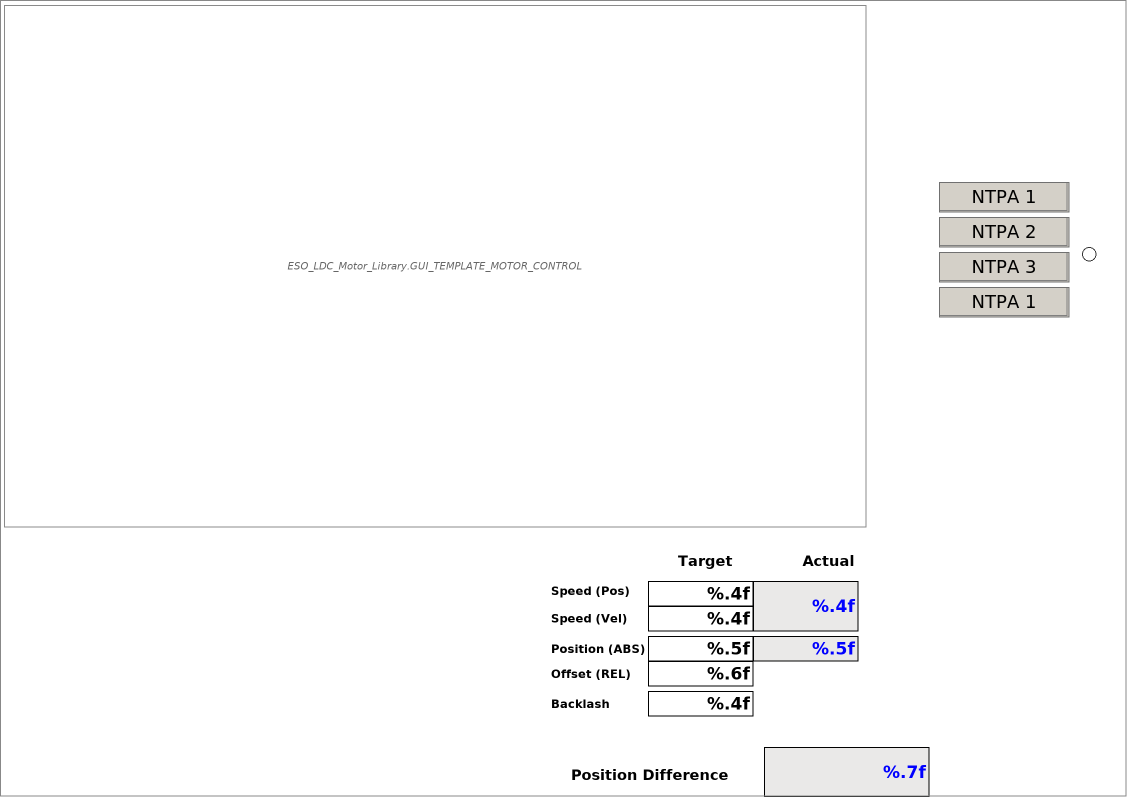
VISUALIZATION GUI_NOTT_TIP_A_CTRL  // 1127x797
    Frame (4,5 862x522)
        shows ESO_LDC_Motor_Library.GUI_TEMPLATE_MOTOR_CONTROL(m_Instance := MAIN.nott_ics.TipTilt.ptrTipActuatorsA[MAIN.nott_ics.TipTilt.guiTipActuatorsAIndex]^)
    Rectangle (548,581 95x20), "Speed (Pos)"
    Rectangle (753,636 105x25), "%.5f", text variable: MAIN.nott_ics.Delay_Lines.ptrDelayLines[MAIN.nott_ics.Delay_Lines.guiShutterIndex]^.stat.lrPosActual, input disabled if: false
    Rectangle (675,551 190x20), "Target Actual"
    Rectangle (548,639 95x20), "Position (ABS)"
    Rectangle (753,581 105x50), "%.4f", text variable: MAIN.nott_ics.Delay_Lines.ptrDelayLines[MAIN.nott_ics.Delay_Lines.guiShutterIndex]^.stat.lrVelActual, input disabled if: false
    Rectangle (648,606 105x25), "%.4f", text variable: MAIN.nott_ics.Delay_Lines.ptrDelayLines[MAIN.nott_ics.Delay_Lines.guiShutterIndex]^.ctrl.lrVelocity
        OnMouseDown: write the text variable via Default
    Rectangle (548,694 95x20), "Backlash"
    Rectangle (648,691 105x25), "%.4f", text variable: MAIN.nott_ics.Delay_Lines.ptrDelayLines[MAIN.nott_ics.Delay_Lines.guiShutterIndex]^.cfg.lrBacklash
        OnMouseDown: write the text variable via Default
    Rectangle (548,606 95x25), "Speed (Vel)"
    Rectangle (648,636 105x25), "%.5f", tooltip "Absolute position used by "MOVE ABS"", text variable: MAIN.nott_ics.Delay_Lines.ptrDelayLines[MAIN.nott_ics.Delay_Lines.guiShutterIndex]^.ctrl.lrPosition
        OnMouseDown: write the text variable via Default
    Rectangle (648,581 105x25), "%.4f", text variable: MAIN.nott_ics.Delay_Lines.ptrDelayLines[MAIN.nott_ics.Delay_Lines.guiShutterIndex]^.cfg.lrDefaultVelocity
        OnMouseDown: write the text variable via Default
    Rectangle (548,664 95x20), "Offset (REL)"
    Rectangle (648,661 105x25), "%.6f", tooltip "Relative offset used by "MOVE REL"", text variable: MAIN.nott_ics.Delay_Lines.ptrDelayLines[MAIN.nott_ics.Delay_Lines.guiShutterIndex]^.ctrl.lrOffset
        OnMouseDown: write the text variable via Default
    Rectangle (764,747 165x50), "%.7f", text variable: MAIN.nott_ics.Delay_Lines.ptrDelayLines[MAIN.nott_ics.Delay_Lines.guiShutterIndex]^.stat.lrPosError, input disabled if: false
    Rectangle (568,765 190x20), "Position Difference"
    RadioButton (1080,184 47x140), variable: MAIN.nott_ics.TipTilt.guiTipActuatorsAIndex-1
        Areas[0]: Text=Radiobutton
        Areas[1]: Text=Radiobutton
    Button (939,182 130x30), "NTPA 1"
        OnMouseClick: execute { MAIN.nott_ics.TipTilt.guiTipActuatorsAIndex := 1; }
    Button (939,217 130x30), "NTPA 2"
        OnMouseClick: execute { MAIN.nott_ics.TipTilt.guiTipActuatorsAIndex := 2; }
    Button (939,252 130x30), "NTPA 3"
        OnMouseClick: execute { MAIN.nott_ics.TipTilt.guiTipActuatorsAIndex := 3; }
    Button (939,287 130x30), "NTPA 1"
        OnMouseClick: execute { MAIN.nott_ics.TipTilt.guiTipActuatorsAIndex := 4; }
END_VISUALIZATION

(* stored: Version 1.1.0.1, ProductVersion 3.1.4024.12
   Visu GUI_NOTT_TIP_A_CTRL: Id {f3bbbd92-f3f0-46b3-ac91-97484ac21769} *)
